TYPE Point2D :
STRUCT
	X : LREAL;
	Y : LREAL;
END_STRUCT
END_TYPE

(* stored: Version 1.1.0.1
   DUT Point2D: Id {c44b1d0a-9ad3-0719-394c-edf5808a0a9f} *)
